//
// Evacuation System Controller.
// The system consists of:
// - Evacuation Valve
// - Root Pump
// - Turbo Pump
//
FUNCTION_BLOCK FB_CRYO_EVACUATION_SYSTEM
VAR_INPUT
	in_Cryo_Cfg:			T_CRYO_CFG;					// Cryo configuration
	in_Temp_Cryo:			T_CRYO_TEMPERATURE_STATUS;	// Cold Bench temperature	
	in_Pressure_Cryo:		T_CRYO_PRESSURE_STATUS;		// Cryostat Pressure
	in_Pressure_Evac:		T_CRYO_PRESSURE_STATUS;		// Evacuation Pressure
	
	in_bRepressValveOpen:	BOOL;	// Repressure Valve Open flag
	in_bRepressValveOK:		BOOL;	// Repressure Valve OK flag
	in_nFeedback:	E_CRYO_BIN_ACT_FEEDBACK := E_CRYO_BIN_ACT_FEEDBACK.ON_ONLY;	// Feedbacks
	// Time between closing Vac valve and Switching OFF the vac Pump [ms]
	in_nTimeout:	UDINT := 3200;	// Timeout for switching on/off [ms]
	in_bEnable:		BOOL := FALSE;	// Controller active while in_bEnable is TRUE
	in_bCmd:		BOOL := FALSE;	// ON=TRUE, OFF=FALSE
END_VAR
VAR
	
	{attribute 'OPC.UA.DA' := '0'}
	i_bRootPumpOn	AT%I*:	BOOL;		// Root Pump Feedback
	{attribute 'OPC.UA.DA' := '0'}
	i_bTurboPumpOn	AT%I*:	BOOL;		// Turbo Pump Feedback
	
	{attribute 'OPC.UA.DA' := '0'}
	q_bPumpCtrl		AT%Q*:	BOOL;			// Pump Control signal
	
	stat:			T_CRYO_EVACUATION_SYSTEM_STATUS;

	{attribute 'OPC.UA.DA' := '1'}
	Valve:	FB_CRYO_BIN_ACT;			// Evacuation Valve 

	{attribute 'OPC.UA.DA' := '0'}
	bExecute_Valve:	BOOL := FALSE;

	{attribute 'OPC.UA.DA' := '0'}
	nCommand_Valve:	E_CRYO_BIN_ACT_CMD	:= E_CRYO_BIN_ACT_CMD.NONE;	// Command

	{attribute 'OPC.UA.DA' := '0'}
	bReset:		BOOL := FALSE;		// RESET Command

	{attribute 'OPC.UA.DA' := '0'}
	bValveCmd:	BOOL := FALSE;		// Valve Command - TRUE=OPEN, FALSE=CLOSE


	{attribute 'OPC.UA.DA' := '0'}
	timerTurbo:	TON;		// Timer for Turbo Pump
	
	{attribute 'OPC.UA.DA' := '0'}
	timerValveDelay:	TON;		// Timer for measuring time after Valve is closed
	
	{attribute 'OPC.UA.DA' := '0'}
	timerValveCtrl:	TON;		// Timer for Valve open/close timeout
	
	{attribute 'OPC.UA.DA' := '0'}
	trigEnable:	R_TRIG;			// Trigger for in_bEnable
	
	{attribute 'OPC.UA.DA' := '0'}
	trigDisable:F_TRIG;			// Trigger for in_bEnable=FALSE, i.e. Disable
	
	{attribute 'OPC.UA.DA' := '0'}
	trigTurbo:	R_TRIG;		// Trigger for start of TurboPump
	
	{attribute 'OPC.UA.DA' := '0'}
	trigValveClosed:	R_TRIG;		// Trigger for Valve Closed. Start timerValve on trigger.
	
END_VAR

// Increment cycle counter
stat.nCycleCounter := stat.nCycleCounter + 1;

// Pump control based on Valve status.
M_PumpCtrl();

// Check for errors
M_CheckErrors();

// Get Valve Command based on pressure and temperature conditions
M_SetValveCommand();


// Execute Valve FB on every cycle
Valve(	in_bExecute	:= bExecute_Valve,
		in_nCommand	:= nCommand_Valve,
		in_nFeedback:= in_nFeedback);


M_StateMachine();

METHOD M_CheckErrors
VAR_INPUT
END_VAR
VAR
END_VAR
// TODO: Set stat.sStatus for each failure
IF Valve.stat.bON  AND  (in_bRepressValveOpen  OR  NOT in_bRepressValveOK) THEN
	// Emergency situation. Close the Valve
	stat.bEmergency	:= TRUE;
	stat.bError	:= TRUE;
ELSIF stat.bEnabled  AND  (in_bRepressValveOpen  OR  NOT in_bRepressValveOK) THEN
	// The Evacuation system should never be enabled 
	// if there is a problem with the repressurizing valve.
	// Emergency situation. Do not operate.
	stat.bEmergency	:= TRUE;
	stat.bError	:= TRUE;
ELSIF NOT in_bRepressValveOK THEN
	stat.bError	:= TRUE;
ELSIF NOT in_Pressure_Cryo.bValid THEN
	stat.bError	:= TRUE;
ELSIF NOT in_Pressure_Evac.bValid THEN
	stat.bError	:= TRUE;
ELSIF Valve.stat.bError THEN
	stat.bError	:= TRUE;
ELSE
	stat.bError	:= FALSE;
END_IF

// Additional check for emergency situation.
// If there is an error while the Evacuation Valve is open, close it immediately.
IF stat.bError  AND  Valve.stat.bON  THEN
	stat.bEmergency	:= TRUE;
END_IF

IF stat.bError  THEN
	stat.bEnabled	:= FALSE;	// Disable Evacuation System
END_IF
END_METHOD

// Pump control based on Valve status.
METHOD M_PumpCtrl
VAR_INPUT
END_VAR
//
// Capture in_bEnable going TRUE.
// When it happens, start the pumps by activating the control output.
//
trigEnable(CLK:=in_bEnable);
IF trigEnable.Q THEN
	stat.bEnabled	:= TRUE;
	stat.bEmergency	:= FALSE;	// Clear emergency warning, if any
	stat.bError		:= FALSE;	// Clear error
	q_bPumpCtrl		:= TRUE;	// Start pumps
ELSIF NOT in_bEnable THEN
	stat.bEnabled		:= FALSE;
END_IF


//
// Set the status of the Root Pump
//
stat.bRootPumpON	:= i_bRootPumpOn;


//
// Set the status of the Turbo Pump
//
IF i_bTurboPumpOn THEN
	// Turbo pump is running.
	stat.bTurboPumpON	:= TRUE;
ELSE
	timerTurbo(IN:=FALSE);
	stat.bTurboPumpON		:= FALSE;
	stat.bTurboPump10min	:= FALSE;
END_IF



//
// Capture the moment when Turbo Pump started.
// Turbo Pump is fully operational after 10 min of operation (in_nTime_TurboPump).
//
// Execute timer for Turbo Pump
timerTurbo();

trigTurbo(CLK:=stat.bTurboPumpON);
IF trigTurbo.Q  THEN
	//
	// Turbo Pump has just started.
	// Start the timer that will signal that the turbo pump is fully operational.
	//
	// Reset the timer.
	timerTurbo(IN:=FALSE);
	// Start the timer for Turbo Pump warmup.
	timerTurbo(IN:=TRUE,PT:=UDINT_TO_TIME(in_Cryo_Cfg.nTime_TurboPump));
END_IF

IF timerTurbo.Q THEN
	// Turbo Pump is now fully operational.
	stat.bTurboPump10min	:= TRUE;
END_IF


//
// Capture the moment when the Valve is closed or the system is disabled.
// Pumps should be stopped in_nTime_DeltaTValve [ms] (e.g. 2000ms) after this event.
//
// Execute timer for Valve timer
timerValveDelay();


//
// Capture the moment when the valve is closed.
// Start the delay timer for in_Cryo_Cfg.nTime_DeltaTValve ms.
// After the delay, it is safe to stop the pumps.
//
trigValveClosed(CLK:=NOT stat.bValveOpen);
trigDisable(CLK:=stat.bEnabled);	// Falling edge of bEnable
IF trigValveClosed.Q OR trigDisable.Q  THEN
	// Reset the timer
	timerValveDelay(IN:=FALSE);
	// Start the Valve timer.
	timerValveDelay(IN:=TRUE,PT:=UDINT_TO_TIME(in_Cryo_Cfg.nTime_DeltaTValve));
END_IF


//
// The delay timer has expired.
// It is safe to stop the pumps.
//
IF timerValveDelay.Q THEN
	// Reset the timer
	timerValveDelay(IN:=FALSE);
	// Stop the pumps if evacuation is disabled
	IF NOT stat.bEnabled THEN
		q_bPumpCtrl	:= FALSE;
	END_IF
END_IF

// Update output var
stat.bValveOpen	:= Valve.stat.bON;
END_METHOD

METHOD M_SetStatus
VAR_INPUT
	nState:	E_CRYO_EVAC_SYS_STATE;
END_VAR
// TODO: Complete this


CASE nState OF
	
	E_CRYO_EVAC_SYS_STATE.OFF:
	stat.bDone	:= TRUE;
	stat.bBusy	:= FALSE;
	IF NOT stat.bError THEN
		stat.sState	:= 'OFF';
	END_IF
	stat.bActive	:= FALSE;
	
	E_CRYO_EVAC_SYS_STATE.ACTIVE_CLOSED:
	stat.bDone	:= TRUE;
	stat.bBusy	:= FALSE;
	IF NOT stat.bError THEN
		stat.sState	:= 'ACTIVE_OFF';
	END_IF
	stat.bActive	:= TRUE;
	
	E_CRYO_EVAC_SYS_STATE.ACTIVE_OPEN:
	stat.bDone	:= TRUE;
	stat.bBusy	:= FALSE;
	stat.bError	:= FALSE;
	stat.bActive	:= TRUE;
	stat.sState	:= 'ACTIVE_ON';
	
	E_CRYO_EVAC_SYS_STATE.ACTIVE_OPENING:
	stat.bDone	:= FALSE;
	stat.bBusy	:= TRUE;
	stat.bError	:= FALSE;
	stat.bActive	:= TRUE;
	stat.sState	:= 'ACTIVE_SWITCHING_ON...';
	
	E_CRYO_EVAC_SYS_STATE.ACTIVE_CLOSING:
	stat.bDone	:= FALSE;
	stat.bBusy	:= TRUE;
	stat.bError	:= FALSE;
	stat.bActive	:= TRUE;
	stat.sState	:= 'ACTIVE_SWITCHING_OFF...';
	
	E_CRYO_EVAC_SYS_STATE.ERROR:
	stat.bDone	:= TRUE;
	stat.bBusy	:= FALSE;
//	stat.bError	:= TRUE;
	stat.bActive	:= FALSE;
//	stat.sState	:= 'ERROR';

END_CASE
END_METHOD

//
// Determines if the valve should be open or closed.
// It sets the internal variable nCommand_Valve.
//
METHOD M_SetValveCommand
VAR_INPUT
END_VAR
// Reset bExecute_Valve flag and the Valve command.
// They might be set again depending on the bEnable flag and the environmental conditions.
bExecute_Valve	:= FALSE;
nCommand_Valve	:= E_CRYO_BIN_ACT_CMD.NONE;


// 
// Set the Valve command based on temperature and pressure.
// If the system is not enabled or there is an error, the valve should be closed.
//
IF stat.bError THEN
	// Close the Valve on any error.
	nCommand_Valve	:= E_CRYO_BIN_ACT_CMD.OFF;
ELSIF NOT stat.bEnabled THEN
	// Close the Valve if the system is Disabled/OFF.
	nCommand_Valve	:= E_CRYO_BIN_ACT_CMD.OFF;
ELSIF 	(in_Pressure_Cryo.lrPressure > in_Cryo_Cfg.lrPress_Atm)  AND  
		(in_Temp_Cryo.lrTempK > in_Cryo_Cfg.lrTemp_Warm) THEN
	// Cryo is Warm and Pressurized - safe to open Valve.
	nCommand_Valve	:= E_CRYO_BIN_ACT_CMD.ON;
//ELSIF NOT in_Pressure_Cryo.bInVacuum THEN
ELSIF in_Pressure_Cryo.lrPressure >= in_Cryo_Cfg.lrPress_InVac THEN
	// If not in vacuum, it means the cryostat must be WARM.
	IF (in_Pressure_Evac.lrPressure < in_Pressure_Cryo.lrPressure) THEN
		nCommand_Valve	:= E_CRYO_BIN_ACT_CMD.ON;
	END_IF
ELSIF in_Temp_Cryo.lrTempK < in_Cryo_Cfg.lrTemp_Precooled THEN
	// Cryostat is COLD.
	IF ((in_Pressure_Evac.lrPressure < in_Pressure_Cryo.lrPressure) AND stat.bTurboPumpON) OR  
		(stat.bTurboPump10min AND in_Pressure_Evac.lrPressure < 7.0E-5) THEN
		nCommand_Valve	:= E_CRYO_BIN_ACT_CMD.ON;
	END_IF
//ELSIF in_Pressure_Cryo.bInVacuum THEN
ELSIF in_Pressure_Cryo.lrPressure < in_Cryo_Cfg.lrPress_InVac THEN
	// Cryostat is in vacuum.
	IF (in_Pressure_Evac.lrPressure < in_Pressure_Cryo.lrPressure)  AND stat.bTurboPumpON THEN
		nCommand_Valve	:= E_CRYO_BIN_ACT_CMD.ON;
	END_IF
END_IF


//
// Apply Valve command depending on the Evacuation System state.
// Update the State as well.
//
IF (stat.bError OR stat.bEmergency) AND stat.nState	<> E_CRYO_EVAC_SYS_STATE.ACTIVE_CLOSING THEN
	//
	// There is an error or emergency in the system. 
	// Close the valve. 
	//
	// Trigger Valve closing
	bExecute_Valve	:= TRUE;
	nCommand_Valve	:= E_CRYO_BIN_ACT_CMD.OFF;
	Valve(in_bExecute	:= FALSE);
	Valve(in_bExecute	:= TRUE, in_nCommand := nCommand_Valve);
	stat.nState	:= E_CRYO_EVAC_SYS_STATE.ACTIVE_CLOSING;
ELSIF stat.nState = E_CRYO_EVAC_SYS_STATE.ACTIVE_CLOSED  THEN 
	IF  nCommand_Valve = E_CRYO_BIN_ACT_CMD.ON THEN
		bExecute_Valve	:= TRUE;
		timerValveCtrl(IN:=FALSE);
		timerValveCtrl(IN:=TRUE, PT:=UDINT_TO_TIME(in_nTimeout));
		stat.nState	:= E_CRYO_EVAC_SYS_STATE.ACTIVE_OPENING;
	ELSE
		bExecute_Valve	:= FALSE;
		IF stat.bEnabled THEN
			stat.nState	:= E_CRYO_EVAC_SYS_STATE.ACTIVE_CLOSED;
		ELSE
			stat.nState	:= E_CRYO_EVAC_SYS_STATE.OFF;
		END_IF
	END_IF
ELSIF stat.nState	= E_CRYO_EVAC_SYS_STATE.ACTIVE_OPEN  THEN 
	IF  nCommand_Valve = E_CRYO_BIN_ACT_CMD.OFF  OR  NOT stat.bEnabled  THEN
		bExecute_Valve	:= TRUE;
		timerValveCtrl(IN:=FALSE);
		timerValveCtrl(IN:=TRUE, PT:=UDINT_TO_TIME(in_nTimeout));
		stat.nState	:= E_CRYO_EVAC_SYS_STATE.ACTIVE_CLOSING;
	ELSE
		bExecute_Valve	:= FALSE;
		stat.nState	:= E_CRYO_EVAC_SYS_STATE.ACTIVE_OPEN;
	END_IF
END_IF
END_METHOD

METHOD M_StateMachine
VAR_INPUT
END_VAR
CASE stat.nState OF
	/////////////////////////////////
	E_CRYO_EVAC_SYS_STATE.NONE:
	/////////////////////////////////
	//
	// This is the state on power-up.
	// Determine the initial state based on the command and actuator state.
	IF NOT stat.bEnabled THEN
		IF Valve.stat.bOFF  AND  NOT stat.bRootPumpON AND NOT stat.bTurboPumpON THEN
			stat.nState	:= E_CRYO_EVAC_SYS_STATE.OFF;
		END_IF
	ELSE
		IF	stat.bError	THEN
			IF Valve.stat.bON THEN
				stat.nState	:= E_CRYO_EVAC_SYS_STATE.EMERGENCY;
			ELSE
				stat.nState	:= E_CRYO_EVAC_SYS_STATE.ERROR;
			END_IF
			stat.nState	:= E_CRYO_EVAC_SYS_STATE.ERROR;
		ELSIF Valve.stat.bON THEN
			stat.nState	:= E_CRYO_EVAC_SYS_STATE.ACTIVE_OPEN;
		ELSIF Valve.stat.bOFF  THEN
			stat.nState	:= E_CRYO_EVAC_SYS_STATE.ACTIVE_CLOSED;
		END_IF
	END_IF
	M_SetStatus(stat.nState);	
	RETURN;
	

	/////////////////////////////////
	E_CRYO_EVAC_SYS_STATE.OFF:
	/////////////////////////////////
	//
	IF stat.bEnabled  THEN
		// Set next state.
		stat.nState	:= E_CRYO_EVAC_SYS_STATE.ACTIVE_CLOSED;
	END_IF
	M_SetStatus(stat.nState);	
	RETURN;
	
	
	////////////////////////////////////////
	E_CRYO_EVAC_SYS_STATE.ACTIVE_CLOSING:
	////////////////////////////////////////
	//
	timerValveCtrl();
	IF timerValveCtrl.Q THEN
		// Closing failure
		stat.bCtrlOK	:= FALSE;
		stat.sStatus	:= 'Valve failed to close';
		stat.bError	:= TRUE;
		stat.nState	:= E_CRYO_EVAC_SYS_STATE.ERROR;
	ELSIF NOT stat.bValveOpen THEN
		timerValveCtrl(IN:=FALSE);
		// Set next state.
		stat.nState	:= E_CRYO_EVAC_SYS_STATE.ACTIVE_CLOSED;
	END_IF
	M_SetStatus(stat.nState);	
	RETURN;
	
	
	////////////////////////////////////////
	E_CRYO_EVAC_SYS_STATE.ACTIVE_CLOSED:
	////////////////////////////////////////
	//
	IF	NOT stat.bEnabled  THEN
		// Set next state
		stat.nState	:= E_CRYO_EVAC_SYS_STATE.OFF;
	ELSIF stat.bValveOpen THEN
		// Set next state.
		stat.nState	:= E_CRYO_EVAC_SYS_STATE.ACTIVE_OPEN;
	END_IF
	M_SetStatus(stat.nState);	
	RETURN;
	
	
	////////////////////////////////////////
	E_CRYO_EVAC_SYS_STATE.ACTIVE_OPENING:
	////////////////////////////////////////
	//
	timerValveCtrl();
	IF timerValveCtrl.Q THEN
		// Closing failure
		stat.bCtrlOK	:= FALSE;
		stat.sStatus	:= 'Valve failed to open';
		stat.bError	:= TRUE;
		stat.nState	:= E_CRYO_EVAC_SYS_STATE.ERROR;
	ELSIF stat.bValveOpen THEN
		timerValveCtrl(IN:=FALSE);
		// Set next state.
		stat.nState	:= E_CRYO_EVAC_SYS_STATE.ACTIVE_OPEN;
	END_IF
	M_SetStatus(stat.nState);	
	RETURN;
	
	
	//////////////////////////////////////////
	E_CRYO_EVAC_SYS_STATE.ACTIVE_OPEN:
	//////////////////////////////////////////
	//
	IF NOT stat.bValveOpen THEN
		// Set next state.
		stat.nState	:= E_CRYO_EVAC_SYS_STATE.ACTIVE_CLOSED;
	END_IF
	M_SetStatus(stat.nState);	
	RETURN;
	

	///////////////////////////////////////////
	E_CRYO_EVAC_SYS_STATE.EMERGENCY:
	///////////////////////////////////////////
	//
	IF Valve.stat.bOFF THEN
		// The actuator is OFF, transition completed.
		// Goto Active_Off.
		stat.nState	:= E_CRYO_EVAC_SYS_STATE.ACTIVE_CLOSED;
	END_IF
	M_SetStatus(stat.nState);	
	RETURN;
	
	/////////////////////////////////
	E_CRYO_EVAC_SYS_STATE.ERROR:
	/////////////////////////////////
	//
	M_User_TryRecovery();

END_CASE
END_METHOD

METHOD M_TrgValveClosure : BOOL
VAR_INPUT
END_VAR
END_METHOD

METHOD M_User_TryRecovery
VAR_INPUT
END_VAR
// TODO USER
// This is the default recovery routine.
// To be customided by the user, if needed.
//
IF bReset THEN
	// RESET the controller in order to try to clear error
	bReset	:= FALSE;	// Clear RESET flag
	
	// Trigger action
	Valve(in_bExecute:=FALSE);
	Valve(in_bExecute:=TRUE, in_nCommand:=E_CRYO_BIN_ACT_CMD.OFF);
	
	// Goto SWITCHING_OFF state
	stat.nState	:= E_CRYO_EVAC_SYS_STATE.ACTIVE_CLOSING;
	M_SetStatus(stat.nState);	
ELSIF NOT Valve.stat.bError AND stat.bCtrlOK  THEN
	// Self recovery since everything seems to be OK now.
	// Goto NONE state.
	// From there proper state will be found and set.
	stat.nState	:= E_CRYO_EVAC_SYS_STATE.NONE;
	M_SetStatus(stat.nState);	
END_IF
END_METHOD

END_FUNCTION_BLOCK

(* stored: Version 1.1.0.1, ProductVersion 3.1.4024.9
   POU FB_CRYO_EVACUATION_SYSTEM: Id {3a5b4b27-7f89-4008-be6d-bf7a09a5b7ad}, SpecialFunc None
   Method M_CheckErrors: Id {58dbdb83-37fb-45ac-99a0-3e2b7ddf2bbb}
   Method M_PumpCtrl: Id {17f9ea11-2824-4193-b10b-a821d2e435e3}
   Method M_SetStatus: Id {4df05ad5-8278-4f54-b5f4-4c2d99497b64}
   Method M_SetValveCommand: Id {548f543d-7acd-4484-a57d-4f54716e6ed7}
   Method M_StateMachine: Id {ea15b5d4-c035-42bd-a71e-59771f61f8ca}
   Method M_TrgValveClosure: Id {17f1425d-8dde-4c31-a85f-f9b73461252b}
   Method M_User_TryRecovery: Id {207ebf33-5778-4baf-9998-80ec070d5d31} *)
